(*
SPDX-FileCopyrightText: Â© 2026 Oleksandr Tiutyk <trofimich@gmail.com>
SPDX-License-Identifier: MIT
License: https://opensource.org/license/mit
*)

(*!
<summary>Provides shared singleton instances of child critical error handling policies.</summary>
*)

{attribute 'no_explicit_call' := 'do not call this function block directly'}
PROGRAM ChildCriticalErrorHandlingPolicies
VAR
	{attribute 'hide'} 
	_ClassName : STRING := __POUNAME();
	
	{attribute 'hide'} 
	_SetErrorAndStop : SetErrorAndStopAfterCriticalChildErrorHandlingPolicy; 
	{attribute 'hide'} 
	_SetErrorAndContinue : SetErrorAndContinueAfterChildCriticalErrorHandlingPolicy; 
	{attribute 'hide'} 
	_Ignore : IgnoreChildCriticalErrorHandlingPolicy; 
END_VAR

(*!
<summary>Gets the class name of the program.</summary>
*)
{attribute 'monitoring' := 'call'}
PROPERTY ClassName : REFERENCE TO STRING
GET
ClassName REF= _ClassName;
END_GET
END_PROPERTY

(*!
<summary>Gets a shared instance of the ignore error policy.</summary>
*)
{attribute 'monitoring' := 'call'}
PROPERTY Ignore : IChildCriticalErrorHandlingPolicy
GET
Ignore := _Ignore;
END_GET
END_PROPERTY

(*!
<summary>Gets the namespace of the program.</summary>
*)
{attribute 'monitoring' := 'call'}
PROPERTY NamespaceName : REFERENCE TO STRING
GET
NamespaceName REF= CurrentNamespace.Name;
END_GET
END_PROPERTY

(*!
<summary>Gets a shared instance of the set error and continue policy.</summary>
*)
{attribute 'monitoring' := 'call'}
PROPERTY SetErrorAndContinue : IChildCriticalErrorHandlingPolicy
GET
SetErrorAndContinue := _SetErrorAndContinue;
END_GET
END_PROPERTY

(*!
<summary>Gets a shared instance of the set error and stop policy.</summary>
*)
{attribute 'monitoring' := 'call'}
PROPERTY SetErrorAndStop : IChildCriticalErrorHandlingPolicy
GET
SetErrorAndStop := _SetErrorAndStop;
END_GET
END_PROPERTY

END_PROGRAM

(* stored: Version 1.1.0.1
   POU ChildCriticalErrorHandlingPolicies: Id {55f93cbf-538f-4156-b101-0a16be141b3c}, SpecialFunc None
   Property ClassName: Id {411cd22a-9274-4d3a-8c7f-29ea3684a9ea}
   Get Get: Id {2ed13241-152a-4988-b4a6-27136b1cacd6}
   Property Ignore: Id {267ef87b-ef80-44fe-b855-8b277a33fdc5}
   Get Get: Id {93458cd1-2bd8-40d3-82a6-73715c944652}
   Property NamespaceName: Id {79889f58-c974-4177-a610-167e9105708f}
   Get Get: Id {417c5e19-1981-4d8e-88a4-673b7ea4ac89}
   Property SetErrorAndContinue: Id {96b0c083-8362-4667-a3fb-758df3b2564f}
   Get Get: Id {a21d2f27-bed2-4645-b944-86e90a4567fd}
   Property SetErrorAndStop: Id {805e0225-c26c-4bb9-991f-8d5ee00adc4a}
   Get Get: Id {e14074a4-3731-48ad-ab47-497f8f34cacd} *)
